# EPICS substitutions: ATCACommonApp/Db/StreamUshort.substitutions
file "streamWf.db"  {
    pattern {      PORT,   DEVICE,    WIDTH,  N,   TYPE,                DTYP,      FTVL,       NELM,    TSE      }
            { "$(PORT)", "$(DEV)",  "Int16", 0, "USHORT", "asynInt16ArrayOut",   "USHORT",  "$(NELM)", "$(TSE)"    }
            { "$(PORT)", "$(DEV)",  "Int16", 1, "USHORT", "asynInt16ArrayOut",   "USHORT",  "$(NELM)", "$(TSE)"    }
            { "$(PORT)", "$(DEV)",  "Int16", 2, "USHORT", "asynInt16ArrayOut",   "USHORT",  "$(NELM)", "$(TSE)"    }
            { "$(PORT)", "$(DEV)",  "Int16", 3, "USHORT", "asynInt16ArrayOut",   "USHORT",  "$(NELM)", "$(TSE)"    }

}
